PROGRAM AUTO_SCREWING
VAR
END_VAR

END_PROGRAM

(* stored: Version 1.1.0.1, ProductVersion 3.1.4022.18
   POU AUTO_SCREWING: Id {a75a531f-4639-40ff-9871-b763ff98fbc9}, SpecialFunc None *)
